TEXTLIST AxisGroupStateList
  0 = 'AxisGroupIdle'
  1 = 'AxisGroupInitialization'
  2 = 'AxisGroupDisabled'
  3 = 'AxisGroupPreStandby'
  4 = 'AxisGroupStandby'
  5 = 'AxisGroupManualMoving'
  6 = 'AxisGroupPreContinuousMoving'
  7 = 'AxisGroupContinuousMoving'
  8 = 'AxisGroupLimitViolation'
  9 = 'AxisGroupEmergency'
  10 = 'AxisGroupFault'
  11 = 'AxisGroupRecovery'
   = ''
END_TEXTLIST

(* stored: Version 1.1.0.1, ProductVersion 3.1.4024.12
   TextList AxisGroupStateList: Id {f8e3457e-2621-4edb-8d39-de9a691b781a} *)
